RoboDK station: Concept_1.rdk

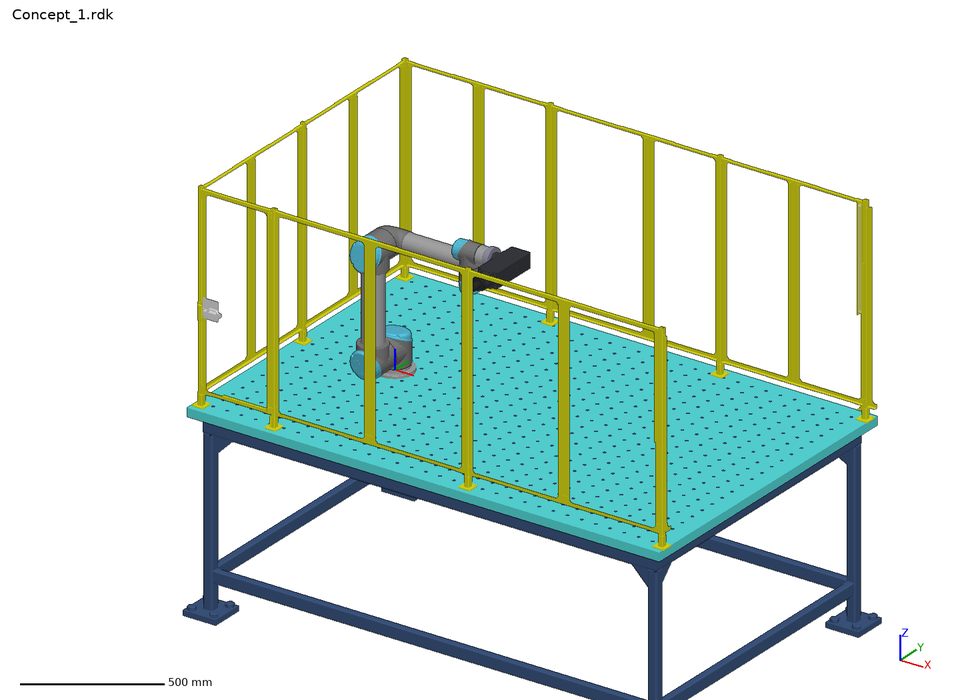
[picture v0: the station drawn from its stored meshes, robots at their saved joint values, targets as dots, program paths as lines]
Station Concept_1 (saved by RoboDK 5.3.4). Poses are relative to the parent item; angles as X-Y-Z fixed-axis rotations.
  - frame UR5 Base at (0, 0, 0) mm
    - robot UR5: 6 axes, payload 5 kg, reach 850 mm, repeatability 0.1 mm, weight 18.4 kg
        modified DH rows (alpha deg, a mm, theta deg, d mm): 0, 0, 0, 89.2; 90, 0, 180, 0; 0, 425, 0, 0; 0, 392.43, 0, 109; -90, 0, 0, 93.65; 90, 0, 180, 82
        joint limits [-360, -360, -360, -360, -360, -360] to [360, 360, 360, 360, 360, 360]; home [0, -90, -90, 0, 90, 0]; saved at [0, -90, -90, 0, 90, 0]
      - tool Spindle, TCP at (278.6, 0, 88) mm, rotated rx 0 ry 90 rz 0 deg, size 85 x 346.5 x 128 mm
  - frame Work Space at (0, 0, 0) mm
    - object Cell Frame 3.5m at (0, 0, 0) mm, size 2018.1 x 1282.7 x 844.7 mm, geometry from Cell-Frame-3.5m.sld
    - object Table 2000x1200x800 at (0, 0, 0) mm, size 2020 x 1340 x 800 mm, geometry from Table-2000mmx1200mmx800mm.sld
  - frame Tube at (0, 0, 0) mm
